TYPE ST_GetBoxInfo :
STRUCT
		//儲位
 		Storgerinfo		:INT; //1~400
		//軌道順序	
		Boxorder		:INT;//1~10
		//放的位置  
		Area  			:E_Location; 
END_STRUCT
 END_TYPE

(* stored: Version 1.1.0.1, ProductVersion 3.1.4024.13
   DUT ST_GetBoxInfo: Id {c116573f-80f0-42c2-8606-46bdd95f286e} *)
